{attribute 'GeneratedUsingTerminal: IODEVICETYPE_ETHERCATPROT'}
{attribute addProperty BoxType "IODEVICETYPE_ETHERCATPROT"}
{attribute addProperty Id "ObjectIdAT %I*DWORD4StateAT %I*UINT2SlaveCountAT %I*UINT2"}
{attribute addProperty CRC "2252992235"}
{attribute addProperty Size "8"}
TYPE InfoData_8649EEEB EXTENDS InputBase_8311D824 :
STRUCT
	{attribute addProperty Name "ObjectId"}
	ObjectId AT %I* : DWORD;
	{attribute addProperty Name "State"}
	State AT %I* : UINT;
	{attribute addProperty Name "SlaveCount"}
	SlaveCount AT %I* : UINT;
END_STRUCT
END_TYPE

(* stored: Version 1.1.0.1, ProductVersion 3.1.4024.12
   DUT InfoData_8649EEEB: Id {6966b683-5851-0651-13d5-0f10e24a478d} *)
